{attribute addProperty BoxType "EPP3744-0041-0016"}
{attribute addProperty Id "DIG_InputsAT %I*DIG_Inputs_0CBA0B4A4860AI_Inputs_ChannelAT %I*ARRAY[0..3] OF AI_Inputs_Channel_5C824630192240DEV_Inputs_DeviceAT %I*DEV_Inputs_Device_1D7635CD4050DIG_OutputsAT %Q*DIG_Outputs_0221D8A31620DEV_Outputs_DeviceAT %Q*DEV_Outputs_Device_2D2EEEA1810WcStateAT %I*WcState_F855686C1620InfoDataAT %I*InfoData_BC63D37F80100"}
{attribute addProperty CRC "1502454832"}
{attribute addProperty SizeInBites "400"}
{attribute addProperty SizeInBytes "50"}
TYPE EPP3744_38AF8BFB :
STRUCT
	{attribute addProperty Name "DIG_Inputs"}
	DIG_Inputs : DIG_Inputs_0CBA0B4A;
	{attribute addProperty Name "AI_Inputs_Channel"}
	AI_Inputs_Channel : ARRAY[0..3] OF AI_Inputs_Channel_5C824630;
	{attribute addProperty Name "DEV_Inputs_Device"}
	DEV_Inputs_Device : DEV_Inputs_Device_1D7635CD;
	{attribute addProperty Name "DIG_Outputs"}
	DIG_Outputs : DIG_Outputs_0221D8A3;
	{attribute addProperty Name "DEV_Outputs_Device"}
	DEV_Outputs_Device : DEV_Outputs_Device_2D2EEEA1;
	{attribute addProperty Name "WcState"}
	WcState : WcState_F855686C;
	{attribute addProperty Name "InfoData"}
	InfoData : InfoData_BC63D37F;
END_STRUCT
END_TYPE

(* stored: Version 1.2.0.0, ProductVersion 3.1.4024.9
   DUT EPP3744_38AF8BFB: Id {ddd9d9ae-77be-40b2-a18d-aa2c429a0f72} *)
